// TIA Portal V19 export
FUNCTION_BLOCK "Alarm_Trigger"   // FB2, LAD
TITLE = Emergency Stop / Alarm
{ S7_Optimized_Access := 'TRUE' }
// Will Hold Info On Alarms and Reset
// stored: MemoryReserve 100, SetENOAutomatically false
   VAR_INPUT
      Alarm_Trigger : Bool;   // Input that Triggers Alarm
      Timer_PT : Time;   // Timer for Trigger Set
      Ack_PB : Bool;   // Acknowledge Alarm Button
      Reset_PB : Bool;   // Reset Alarm Button
   END_VAR
   VAR_OUTPUT
      ALARM : Bool;   // Alarm Status
      ALARM_ACKED : Bool;   // Alarm Acknowledge Status
      ALARM_BLINK : Bool;   // Alarm LED Status
   END_VAR
   VAR
      Alarm_TD : Bool;   // Alarm was Triggered
      Alarm_Active : Bool;   // Alarm is Active
      Alarm_ACK : Bool;   // Alarm was Acknowledged
      Alarm_Reset : Bool;   // Alarm was Reset
      Alarm_Timer { S7_SetPoint := 'True'} : TON_TIME;   // Alarm Timer
   END_VAR
BEGIN

REGION Network 1: Alarm Triggers ( After holding for PTime)
   // Sets Alarm to Triggered after some time.
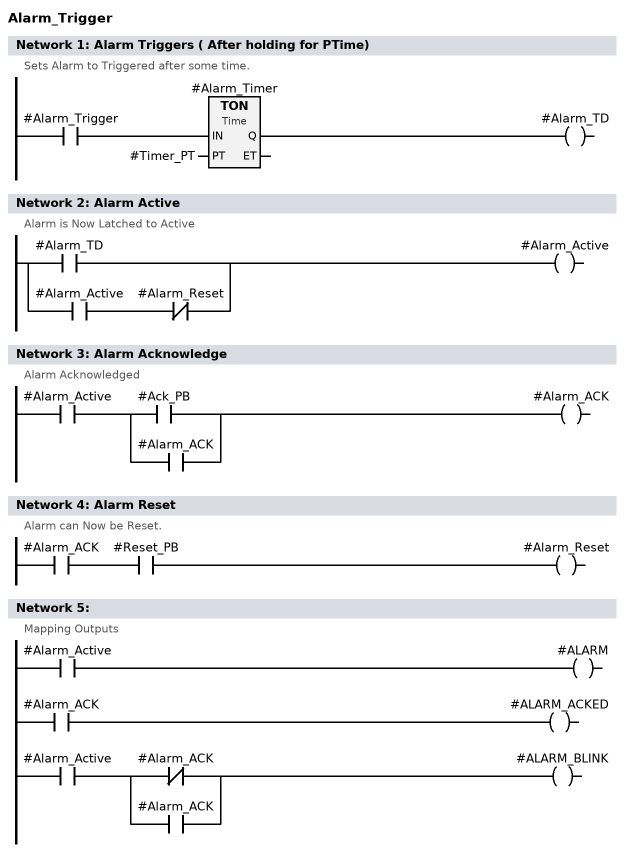
   RUNG wire#powerrail
      Contact( #Alarm_Trigger )
      { S7_Templates := "time_type := Time" } #Alarm_Timer.TON(pt := #Timer_PT, et =>)
      Coil( #Alarm_TD )
   END_RUNG
   // the same network as SCL:
   #Alarm_Timer(IN := #Alarm_Trigger, PT := #Timer_PT);   // TON
   #Alarm_TD := #Alarm_Timer.Q;
END_REGION

REGION Network 2: Alarm Active
   // Alarm is Now Latched to Active
   RUNG wire#powerrail
      Contact( #Alarm_TD )
      wire#w1
      Coil( #Alarm_Active )
   END_RUNG
   RUNG wire#powerrail
      Contact( #Alarm_Active )
      I_Contact( #Alarm_Reset )
   END_RUNG wire#w1
   // the same network as SCL:
   #Alarm_Active := #Alarm_TD OR (#Alarm_Active AND NOT #Alarm_Reset);
END_REGION

REGION Network 3: Alarm Acknowledge
   // Alarm Acknowledged
   RUNG wire#powerrail
      Contact( #Alarm_Active )
      wire#w1
      Contact( #Ack_PB )
      wire#w2
      Coil( #Alarm_ACK )
   END_RUNG
   RUNG wire#w1
      Contact( #Alarm_ACK )
   END_RUNG wire#w2
   // the same network as SCL:
   #Alarm_ACK := #Alarm_Active AND (#Ack_PB OR #Alarm_ACK);
END_REGION

REGION Network 4: Alarm Reset
   // Alarm can Now be Reset.
   RUNG wire#powerrail
      Contact( #Alarm_ACK )
      Contact( #Reset_PB )
      Coil( #Alarm_Reset )
   END_RUNG
   // the same network as SCL:
   #Alarm_Reset := #Alarm_ACK AND #Reset_PB;
END_REGION

REGION Network 5
   // Mapping Outputs
   RUNG wire#powerrail
      Contact( #Alarm_Active )
      Coil( #ALARM )
   END_RUNG
   RUNG wire#powerrail
      Contact( #Alarm_ACK )
      Coil( #ALARM_ACKED )
   END_RUNG
   RUNG wire#powerrail
      Contact( #Alarm_Active )
      wire#w1
      I_Contact( #Alarm_ACK )
      wire#w2
      Coil( #ALARM_BLINK )
   END_RUNG
   RUNG wire#w1
      Contact( #Alarm_ACK )
   END_RUNG wire#w2
   // the same network as SCL:
   #ALARM := #Alarm_Active;
   #ALARM_ACKED := #Alarm_ACK;
   #ALARM_BLINK := #Alarm_Active AND (NOT #Alarm_ACK OR #Alarm_ACK);
END_REGION

REGION Network 6: Spare Network
END_REGION
END_FUNCTION_BLOCK
